      L #s_ISD_ID_Decision.BagIDArray.Decision_Bag_Disposition;
      T #s_Decision_Data.Itm_Data.Process_1.EDS_Decision.Decision_Bag_Disposition;

      L 0;// 0=No decision on current process
      L #s_Decision_Data.Itm_Data.Process_1.EDS_Decision.Decision_Bag_Disposition;
      ==I;
      S #s_Decision_Data.Itm_Data.Process_1.EDS_Decision.No_Decision;
      JC MB10;

      L 1;// 1=Machine alarm
      L #s_Decision_Data.Itm_Data.Process_1.EDS_Decision.Decision_Bag_Disposition;
      ==I;
      S #s_Decision_Data.Itm_Data.Process_1.EDS_Decision.Rejected_Machine;
      JC MB10;

      L 2;// 2=Machine cleared
      L #s_Decision_Data.Itm_Data.Process_1.EDS_Decision.Decision_Bag_Disposition;
      ==I;
      S #s_Decision_Data.Itm_Data.Process_1.EDS_Decision.Cleared_Machine;
      JC MB10;

      L 3;// 3=Machine error / unkown / bag not analyzed
      L #s_Decision_Data.Itm_Data.Process_1.EDS_Decision.Decision_Bag_Disposition;
      ==I;
      S #s_Decision_Data.Itm_Data.Process_1.EDS_Decision.Not_Analyzed;
      JC MB10;

      L 4;// 4=Decision pending
      L #s_Decision_Data.Itm_Data.Process_1.EDS_Decision.Decision_Bag_Disposition;
      ==I;
      S #s_Decision_Data.Itm_Data.Process_1.EDS_Decision.Pending;
      JC MB10;

      L 5;// 5=operator timed out
      L #s_Decision_Data.Itm_Data.Process_1.EDS_Decision.Decision_Bag_Disposition;
      ==I;
      S #s_Decision_Data.Itm_Data.Process_1.EDS_Decision.Timed_Out_Operator;
      JC MB10;

      L 11;//11=operator alarm
      L #s_Decision_Data.Itm_Data.Process_1.EDS_Decision.Decision_Bag_Disposition;
      ==I;
      S #s_Decision_Data.Itm_Data.Process_1.EDS_Decision.Rejected_Operator;
      JC MB10;

      L 12;// 12=operator clear
      L #s_Decision_Data.Itm_Data.Process_1.EDS_Decision.Decision_Bag_Disposition;
      ==I;
      S #s_Decision_Data.Itm_Data.Process_1.EDS_Decision.Cleared_Operator;
      JC MB10;

      L 13;// 13=obvious threat
      L #s_Decision_Data.Itm_Data.Process_1.EDS_Decision.Decision_Bag_Disposition;
      ==I;
      S #s_Decision_Data.Itm_Data.Process_1.EDS_Decision.Obvious_Threat;
      JC MB10;

      L 6;// 6=Machine bag spacing error
      L #s_Decision_Data.Itm_Data.Process_1.EDS_Decision.Decision_Bag_Disposition;
      ==I;
      S #s_Decision_Data.Itm_Data.Process_1.EDS_Decision.Spacing_Error;
      JC MB10;

      L 7;// 7=Forced Reject
      L #s_Decision_Data.Itm_Data.Process_1.EDS_Decision.Decision_Bag_Disposition;
      ==I;
      S #s_Decision_Data.Itm_Data.Process_1.EDS_Decision.Forced_Reject;
      JC MB10;

      SET;// all other result are unknown
      S #s_Decision_Data.Itm_Data.Process_1.EDS_Decision.Not_Analyzed;

MB10:      AN #s_Decision_Data.No_Decision_Expected;
      JCN MB98;

      AN #s_Decision_Data.Valid_LNK_Available;
      JCN MB11;// Item already found, no data reload needed

      A(;
      L #s_Decision_Data.Itm_Data.LNK;
      L 0;
      >I;
      );
      JCN MB12;// If LNK is unknown by EDS, start lookup on pseudo ID

      L #s_Decision_Data.Itm_Data.PEN_ID;
      L "DB_PEN_List".Entries_Present;
      <=I;
      JCN MB98;// If LNK is not in expected range: Abort data attachment

      L "DB_Pending_Record".THIS[#s_Decision_Data.Itm_Data.PEN_ID].PEN_LNK;
      L 0;
      ==I;
      S #s_Decision_Data.No_Decision_Expected;

      AN #s_Decision_Data.No_Decision_Expected;
      JCN MB98;// No HBS record = no screening result expected

      L "DB_Pending_Record".THIS[#s_Decision_Data.Itm_Data.PEN_ID].PEN.LNK;
      L 0;
      >I;
      JCN MB11;

      CALL "FC_Read_ANY_Record"// Read entire LNK record
      (  i_Record_Number             := #s_Decision_Data.Itm_Data.LNK ,
         i_ANY_Data_Record           := "DB_UDT_LNK_Record" ,
         i_ANY_Data                  := #s_Decision_Data.Itm_Data.LNK_Record ,
         i_DB                        := "DB_LNK_List" ,
         i_DB_Event_Num              := #t_DB_Event_Num_Object
      );

MB11:      L #s_Decision_Data.Itm_Data.Pseudo;
      L "DB_Pending_Record".THIS[#s_Decision_Data.Itm_Data.PEN_ID].PEN.PEN_Process_1.Screen_Result.Pseudo_ID;
      ==D;
      JCN MB12;

      L #s_Decision_Data.Itm_Data.PEN_ID;
      L 0;
      >I;
      JCN MB12;

      L "DB_Pending_Record".THIS[#s_Decision_Data.Itm_Data.PEN_ID].PEN.PEN_Process_1.ID_Screening;
      L #i_HBO_ID;
      ==D;
      S #s_Decision_Data.Valid_LNK_Available;
      R #s_Decision_Data.Itm_Data.Process_1.No_Decision_Expected;

      JU MB98;

MB12:      A #s_Decision_Data.Valid_LNK_Available;
      JC MB98;

      A #s_Decision_Data.Itm_Data.Process_1.No_Decision_Expected;
      JC MB99;

      SET;
      S #s_Decision_Data.Inval_LNK_Pseudo_Lookup;

      L DINT#0;
      L #s_Decision_Data.Itm_Data.Pseudo;
      <>D;
      JCN MB98;// If no pseudo available: End bag lookup, else: lookup bag by pseudo

      CALL "FC_PEN_Srch_ID"
      (  i_Pseudo_ID                 := #s_Decision_Data.Itm_Data.Pseudo ,
         o_PEN_ID                    := #s_Decision_Data.Itm_Data.PEN_ID
      );

      L #s_Decision_Data.Itm_Data.PEN_ID;
      L 0;
      >I;
      JCN MB99;

MB50:      AN #s_Decision_Data.Valid_LNK_Available;
      JCN MB98;// If correct LNK not found yet, try next pseudo

MB98:      A #s_Decision_Data.Itm_Data.Process_1.No_Decision_Expected;
      O #s_Decision_Data.No_Decision_Expected;
      AN #s_Decision_Data.Itm_Data.Process_1.EDS_Decision.No_Decision;
      AN #s_Decision_Data.Itm_Data.Process_1.EDS_Decision.Forced_Reject;// We already know the item is no longer present
      AN #s_Decision_Data.Itm_Data.Process_1.EDS_Decision.Not_Analyzed;//With LIC=0 EDS responds Not Analyzed
      JCN MB99;// Unable to find applicable item or item is not pending while decision is present: log event

      CALL "FC_Write_Event"// Screening: Unexpected decision from EDS
      (  i_Message_ID                := 3213 ,
         i_Event_value               := #s_ISD_ID_Decision.BagIDArray.LNK ,
         i_DB_Event_Num              := #t_DB_Event_Num_Object ,
         o_Return_Value              := #t_INT_not_used
      );

MB99:      NOP 0;
NETWORK
TITLE = NA: Upd. PROCESS_1 records (HBS/LIC) upon decision + PackageRep
//Update local bag records to match received decisions
      A #s_OS_New_Decision_Avail;
      A #s_Decision_Data.Valid_LNK_Available;
      JCN NA99;

      AN #s_Decision_Data.Itm_Data.Process_1.No_Decision_Expected;
      JCN NA99;// If no HBS record available: stop receival, else: process

      CALL MOVE
      {value_type := 'Variant'}
      (  IN                          := "DB_Pending_Record".THIS[#s_Decision_Data.Itm_Data.PEN_ID].PEN ,
         OUT                         := #s_Decision_Data.Itm_Data.HBS_Record
      );

      AN #s_Decision_Data.Itm_Data.HBS_Record.PEN_Process_1.Result_Pending;
      O #s_Decision_Data.Itm_Data.HBS_Record.PEN_General.Item_Lost;
      O(;
      L #s_Decision_Data.Itm_Data.HBS_Record.PEN_General.HBA_LNK;
      L #s_Decision_Data.Itm_Data.LNK;
      <>I;
      );
      S #s_Decision_Data.Itm_Data.Process_1.No_Decision_Expected;// No decision expected concluded by HBS record content

      L "DB_Pending_Record".THIS[#s_Decision_Data.Itm_Data.PEN_ID].PEN.LNK;
      L 0;
      ==I;
      S #s_Decision_Data.LIC_Missing;

      A #s_Decision_Data.Itm_Data.Process_1.No_Decision_Expected;
      O #s_Decision_Data.Itm_Data.Process_1.EDS_Decision.No_Decision;
      JC NA23               ;// If process 1 decision expected and present: process, else: make sure PackageReport DB is empty

      A #s_Decision_Data.Itm_Data.Process_1.EDS_Decision.Cleared_Machine;
      AN #s_Decision_Data.Itm_Data.HBS_Record.PEN_Process_1.Machine_Result_Rcvd;
      JCN NA01;
      S #s_Decision_Data.Itm_Data.HBS_Record.PEN_General.Bag_Status.Cleared;
      R #s_Decision_Data.Itm_Data.HBS_Record.PEN_General.Bag_Status.Alarmed;

      L 1;// Update screening status : "CLEAR"
      T #s_Decision_Data.Itm_Data.Process_1.Machine_Result_To_HL;

      SET;
      S #s_Decision_Data.Itm_Data.HBS_Record.PEN_Process_1.Screen_Result.Reached_Screen_Level_1;

      JU NA20;
NA01:      A #s_Decision_Data.Itm_Data.Process_1.EDS_Decision.Rejected_Machine;
      AN #s_Decision_Data.Itm_Data.HBS_Record.PEN_Process_1.Machine_Result_Rcvd;
      JCN NA02;
      S #s_Decision_Data.Itm_Data.HBS_Record.PEN_General.Bag_Status.Alarmed;
      R #s_Decision_Data.Itm_Data.HBS_Record.PEN_General.Bag_Status.Cleared;

      L 2;// Update screening status : "REJECT"
      T #s_Decision_Data.Itm_Data.Process_1.Machine_Result_To_HL;

      SET;
      S #s_Decision_Data.Itm_Data.HBS_Record.PEN_Process_1.Screen_Result.Failed_Screen_Level_1;

      JU NA20;

NA02:      A #s_Decision_Data.Itm_Data.Process_1.EDS_Decision.Not_Analyzed;
      JCN NA04;

      A #s_Decision_Data.Itm_Data.HBS_Record.PEN_General.Bag_Status.NoDecision;
      JCN NA03;
      S #s_Decision_Data.Itm_Data.HBS_Record.PEN_General.Bag_Status.Alarmed;
      R #s_Decision_Data.Itm_Data.HBS_Record.PEN_General.Bag_Status.Cleared;

      L 5;// Suspect
      T #s_Decision_Data.Itm_Data.Process_1.Machine_Result_To_HL;

      SET;
      S #s_Decision_Data.Itm_Data.HBS_Record.PEN_Process_1.Screen_Result.Failed_Screen_Level_1;

      JU NA20;

NA03:      L 5;
      T #s_Decision_Data.Itm_Data.Process_1.Machine_Result_To_HL;

      SET;
      S #s_Decision_Data.Itm_Data.HBS_Record.PEN_General.Bag_Status.Unknown;
//      L     4                    // Not screened/Not Analyzed
//      T     #s_Decision_Data.Itm_Data.HBS_Record.PEN_General.Bag_Status

      JU NA20;

NA04:      A #s_Decision_Data.Itm_Data.Process_1.EDS_Decision.Spacing_Error;
      JCN NA06;

// Check current bag status for result
      A #s_Decision_Data.Itm_Data.HBS_Record.PEN_General.Bag_Status.NoDecision;
      JCN NA05;
      S #s_Decision_Data.Itm_Data.HBS_Record.PEN_General.Bag_Status.Alarmed;
      R #s_Decision_Data.Itm_Data.HBS_Record.PEN_General.Bag_Status.Cleared;

      L 6;
      T #s_Decision_Data.Itm_Data.Process_1.Machine_Result_To_HL;

      SET;
      S #s_Decision_Data.Itm_Data.HBS_Record.PEN_Process_1.Screen_Result.Failed_Screen_Level_1;

      JU NA20;

NA05:      L 5;
      T #s_Decision_Data.Itm_Data.Process_1.Machine_Result_To_HL;

      SET;
      S #s_Decision_Data.Itm_Data.HBS_Record.PEN_General.Bag_Status.Unknown;
//      L     4                    // Not screened/Not Analyzed
//      T     #s_Decision_Data.Itm_Data.HBS_Record.PEN_General.Bag_Status

      JU NA20;

NA06:      A #s_Decision_Data.Itm_Data.Process_1.EDS_Decision.Cleared_Operator;// Evaluate L2 (operator) decision
      AN #s_Decision_Data.Itm_Data.HBS_Record.PEN_Process_1.Operator_Result_Rcvd;
      JCN NA07;// L2 clear
      S #s_Decision_Data.Itm_Data.HBS_Record.PEN_General.Bag_Status.Cleared;
      R #s_Decision_Data.Itm_Data.HBS_Record.PEN_General.Bag_Status.Alarmed;

      L 1;// Update screening status : "CLEAR"
      T #s_Decision_Data.Itm_Data.Process_1.Operator_Result_To_HL;

      SET;
      S #s_Decision_Data.Itm_Data.HBS_Record.PEN_Process_1.Screen_Result.Reached_Screen_Level_2;

      JU NA20;

NA07:      A #s_Decision_Data.Itm_Data.Process_1.EDS_Decision.Rejected_Operator;// L2 fail
      AN #s_Decision_Data.Itm_Data.HBS_Record.PEN_Process_1.Operator_Result_Rcvd;
      JCN NA08;
      S #s_Decision_Data.Itm_Data.HBS_Record.PEN_General.Bag_Status.Alarmed;
      R #s_Decision_Data.Itm_Data.HBS_Record.PEN_General.Bag_Status.Cleared;

      L 6;// Update screening status : "UNCLEARED"
      T #s_Decision_Data.Itm_Data.Process_1.Operator_Result_To_HL;

      SET;
      S #s_Decision_Data.Itm_Data.HBS_Record.PEN_Process_1.Screen_Result.Failed_Screen_Level_2;

      JU NA20;

NA08:      A #s_Decision_Data.Itm_Data.Process_1.EDS_Decision.Timed_Out_Operator;
      AN #s_Decision_Data.Itm_Data.HBS_Record.PEN_Process_1.Operator_Result_Rcvd;
      JCN NA09;
      S #s_Decision_Data.Itm_Data.HBS_Record.PEN_General.Bag_Status.TimeOut;

      L 4;
      T #s_Decision_Data.Itm_Data.Process_1.Operator_Result_To_HL;

      JU NA20;

NA09:      A #s_Decision_Data.Itm_Data.Process_1.EDS_Decision.Pending;
      JCN NA10;// Pending = L1 unclear
      S #s_Decision_Data.Itm_Data.HBS_Record.PEN_General.Bag_Status.Pending;

      L 6;// Update screening status : "UNCLEARED"
      T #s_Decision_Data.Itm_Data.Process_1.Machine_Result_To_HL;

      SET;
      S #s_Decision_Data.Itm_Data.HBS_Record.PEN_Process_1.Screen_Result.Failed_Screen_Level_1;

      JU NA20;

NA10:      A #s_Decision_Data.Itm_Data.Process_1.EDS_Decision.Obvious_Threat;
      AN #s_Decision_Data.Itm_Data.HBS_Record.PEN_Process_1.Operator_Result_Rcvd;
      JCN NA11;// Obvious threat
      S #s_Decision_Data.Itm_Data.HBS_Record.PEN_General.Bag_Status.Alarmed;
      R #s_Decision_Data.Itm_Data.HBS_Record.PEN_General.Bag_Status.Cleared;

      L 6;
      T #s_Decision_Data.Itm_Data.Process_1.Operator_Result_To_HL;

      SET;
      S #s_Decision_Data.Itm_Data.HBS_Record.PEN_Process_1.Screen_Result.Failed_Screen_Level_2;

      JU NA20;

NA11:      A #s_Decision_Data.Itm_Data.Process_1.EDS_Decision.Forced_Reject;
      JCN NA20;// No record updates, only log message

      CALL "FC_Write_Event"// Log: Screening: Force reject on item
      (  i_Message_ID                := 3813 ,
         i_Event_value               := #s_ISD_ID_Decision.BagIDArray.LNK ,
         i_DB_Event_Num              := #t_DB_Event_Num_Object ,
         o_Return_Value              := #t_INT_not_used
      );

      JU NA99;

NA20:      A #s_Decision_Data.Itm_Data.Process_1.EDS_Decision.Cleared_Machine;
      O #s_Decision_Data.Itm_Data.Process_1.EDS_Decision.Rejected_Machine;
      O #s_Decision_Data.Itm_Data.Process_1.EDS_Decision.Not_Analyzed;
      O #s_Decision_Data.Itm_Data.Process_1.EDS_Decision.Spacing_Error;
      O #s_Decision_Data.Itm_Data.Process_1.EDS_Decision.Cleared_Operator;
      O #s_Decision_Data.Itm_Data.Process_1.EDS_Decision.Rejected_Operator;
      O #s_Decision_Data.Itm_Data.Process_1.EDS_Decision.Timed_Out_Operator;
      O #s_Decision_Data.Itm_Data.Process_1.EDS_Decision.Pending;
      O #s_Decision_Data.Itm_Data.Process_1.EDS_Decision.Obvious_Threat;
      JCN NA99;// In case of new data: Update HBS, LIC and send PackageReport

      CALL MOVE
      {value_type := 'Variant'}
      (  IN                          := #s_Decision_Data.Itm_Data.HBS_Record.PEN_Process_1.Screen_Result ,
         OUT                         := "DB_Pending_Record".THIS[#s_Decision_Data.Itm_Data.PEN_ID].PEN.PEN_Process_1.Screen_Result
      );

      CALL MOVE
      {value_type := 'Variant'}
      (  IN                          := #s_Decision_Data.Itm_Data.HBS_Record.PEN_General.Bag_Status ,
         OUT                         := "DB_Pending_Record".THIS[#s_Decision_Data.Itm_Data.PEN_ID].PEN.PEN_General.Bag_Status
      );

      L 0;
      L #s_Decision_Data.Itm_Data.LNK_Record.HBS;
      <I;
      L "DB_HBS_List".Entries_Present;
      <I;
      JCN NA21;

      CALL MOVE
      {value_type := 'Variant'}
      (  IN                          := #s_Decision_Data.Itm_Data.HBS_Record.PEN_General.Bag_Status ,
         OUT                         := "DB_HBS_List".HBS[#s_Decision_Data.Itm_Data.LNK_Record.HBS].PEN_General.Bag_Status
      );

NA21:      A #s_Decision_Data.Itm_Data.HBS_Record.PEN_Process_1.Update_Send;
      JCN NA22               ;// Enable sending of new data if required
      R #s_Decision_Data.Itm_Data.HBS_Record.PEN_Process_1.Update_Send;
      R "DB_Pending_Record".THIS[#s_Decision_Data.Itm_Data.PEN_ID].PEN.PEN_Process_1.Update_Send;

NA22:      CALL "FC_Write_Event"   // Screening pending: Update request from HBO
      (  i_Message_ID                := 3814 ,
         i_Event_value               := #s_Decision_Data.Itm_Data.LNK ,
         i_DB_Event_Num              := #t_DB_Event_Num_Object ,
         o_Return_Value              := #t_INT_not_used
      );

      AN #s_Decision_Data.LIC_Missing;
      JCN NA23;

      CALL "FC_Write_ANY_Record"
      (  i_Record_Number             := #s_Decision_Data.Itm_Data.LNK_Record.LIC ,
         i_ANY_Data_Record           := "DB_UDT_LIC_Record".BIR.Process_1 ,
         i_ANY_Data                  := #s_Decision_Data.Itm_Data.HBS_Record.PEN_Process_1.Screen_Result ,
         i_DB                        := "DB_LIC_List" ,
         i_DB_Event_Num              := #t_DB_Event_Num_Object
      );

      CALL MOVE
      {value_type := 'Variant'}
      (  IN                          := #s_Decision_Data.Itm_Data.HBS_Record.PEN_General.Bag_Status ,
         OUT                         := "DB_LIC_List".LIC[#s_Decision_Data.Itm_Data.LNK_Record.LIC].BIR.Bag_Status
      );

      CALL MOVE
      {value_type := 'Variant'}
      (  IN                          := #s_Decision_Data.Itm_Data.HBS_Record.PEN_Process_1.Screen_Result ,
         OUT                         := "DB_Pending_Record".THIS[#s_Decision_Data.Itm_Data.PEN_ID].PEN.PEN_Process_1.Screen_Result
      );

      CALL MOVE
      {value_type := 'Variant'}
      (  IN                          := #s_Decision_Data.Itm_Data.HBS_Record.PEN_General.Bag_Status ,
         OUT                         := "DB_Pending_Record".THIS[#s_Decision_Data.Itm_Data.PEN_ID].PEN.PEN_General.Bag_Status
      );

NA23:      L #s_Decision_Data.Itm_Data.Process_1.Machine_Result_To_HL;
      L 0;
      >I;
      S #s_Decision_Data.Send_Package_Report;
      R #s_Decision_Data.Package_Report_Sent;
      JCN NA24;
      S "DB_Pending_Record".THIS[#s_Decision_Data.Itm_Data.PEN_ID].PEN.PEN_Process_1.Machine_Result_Rcvd;

      A #s_Decision_Data.Itm_Data.Process_1.EDS_Decision.Not_Analyzed;
      O(;
      A #s_Decision_Data.Itm_Data.Process_1.EDS_Decision.Cleared_Machine;
      AN #s_Decision_Data.Itm_Data.HBS_Record.PEN_Process_1.Screen_Result.Required_Screen_Level_2;
      );
      O #s_Decision_Data.Itm_Data.Process_1.EDS_Decision.Spacing_Error;
      O #s_Decision_Data.Itm_Data.Process_1.EDS_Decision.Forced_Reject;
      JCN NA24;
      R "DB_Pending_Record".THIS[#s_Decision_Data.Itm_Data.PEN_ID].PEN.PEN_Process_1.Result_Pending;

      L #s_Decision_Data.Itm_Data.LNK;
      L 11000;// Bit 11 Process End
      +I;
      T #t_Scn_Event;

      CALL "FC_Write_Event"
      (  i_Message_ID                := 2610 ,
         i_Event_value               := #t_Scn_Event ,
         i_DB_Event_Num              := #t_DB_Event_Num_Object ,
         o_Return_Value              := #t_INT_not_used
      );

NA24:      L #s_Decision_Data.Itm_Data.Process_1.Operator_Result_To_HL;
      L 0;
      >I;
      S #s_Decision_Data.Send_Package_Report;
      R #s_Decision_Data.Package_Report_Sent;
      JCN NA25;
      S "DB_Pending_Record".THIS[#s_Decision_Data.Itm_Data.PEN_ID].PEN.PEN_Process_1.Operator_Result_Rcvd;
      R "DB_Pending_Record".THIS[#s_Decision_Data.Itm_Data.PEN_ID].PEN.PEN_Process_1.Result_Pending;

NA25:      A #s_Decision_Data.Send_Package_Report;
      AN #s_Decision_Data.Package_Report_Sent;
      JCN NA99;

      OPN "DB_Send_FIFO";
      L DBNO;
      T #t_INT_not_used;

      CALL MOVE
      {value_type := 'Variant'}
      (  IN                          := #s_Decision_Data.Itm_Data.HBS_Record.PEN_General.Bag_Status ,
         OUT                         := "DB_Pending_Record".THIS[#s_Decision_Data.Itm_Data.PEN_ID].PEN.PEN_General.Bag_Status
      );

      L "DB_Pending_Record".THIS[#t_PEN_ID].PEN.PEN_General.TRA_LNK;
      L 0;
      <>I;
      JCN NA26;

      CALL "FC_Crt_PendingUpd"
      (  i_ID                        := #i_HBO_ID ,
         i_Data                      := #s_Decision_Data.Itm_Data.PEN_ID ,
         i_TRA_LNK                   := "DB_Pending_Record".THIS[#t_PEN_ID].PEN.PEN_General.TRA_LNK ,
         i_FIFO_PLC_DB_num           := #t_INT_not_used ,
         i_DB_Event_Num              := #t_DB_Event_Num_Object ,
         i_Mess_Type                 := 1
      );

NA26:      AN #s_Decision_Data.LIC_Missing;
      JCN NA97;

      L #s_Decision_Data.Itm_Data.LNK_Record.HBS;
      L 0;
      >I;
      JCN NA97;

      CALL MOVE
      {value_type := 'Variant'}
      (  IN                          := "DB_Pending_Record".THIS[#s_Decision_Data.Itm_Data.PEN_ID].PEN.PEN_General.Bag_Status ,
         OUT                         := "DB_HBS_List".HBS[#s_Decision_Data.Itm_Data.LNK_Record.HBS].PEN_General.Bag_Status
      );

      CALL MOVE
      {value_type := 'Variant'}
      (  IN                          := "DB_Pending_Record".THIS[#s_Decision_Data.Itm_Data.PEN_ID].PEN.PEN_Process_1 ,
         OUT                         := "DB_HBS_List".HBS[#s_Decision_Data.Itm_Data.LNK_Record.HBS].PEN_Process_1
      );

      CALL "FC_Write_ANY_Record"
      (  i_Record_Number             := #s_Decision_Data.Itm_Data.LNK_Record.LIC ,
         i_ANY_Data_Record           := "DB_UDT_LIC_Record".BIR.Process_1 ,
         i_ANY_Data                  := #s_Decision_Data.Itm_Data.HBS_Record.PEN_Process_1.Screen_Result ,
         i_DB                        := "DB_LIC_List" ,
         i_DB_Event_Num              := #t_DB_Event_Num_Object
      );

      CALL "FC_Write_Event"
      (  i_Message_ID                := 1210 , // Send PackageReport: Screening Result
         i_Event_value               := #s_Decision_Data.Itm_Data.LNK ,
         i_DB_Event_Num              := #t_DB_Event_Num_Object ,
         o_Return_Value              := #t_INT_not_used
      );

      JU NA98;

NA97:      CALL "FC_Crt_PackScrnPen"
      (  i_ID                        := #i_HBO_ID ,
         i_PEN_ID                    := #s_Decision_Data.Itm_Data.PEN_ID ,
         i_FIFO_PLC_DB_num           := #t_INT_not_used ,
         i_DB_Event_Num              := #t_DB_Event_Num_Object
      );

NA98:      SET;
      S #s_Decision_Data.Package_Report_Sent;

NA99:      NOP 0;
NETWORK
TITLE = OA: Update PROCESS_1 statisticals upon decision or timeout

      A #s_OS_New_Decision_Avail;
      AN #i_Test_Mode_Active;// Don't update machine decision statisticals in test mode
      JCN OA99;

      A #s_Decision_Data.Itm_Data.Process_1.EDS_Decision.Cleared_Machine;
      JCN OA02;

      L #s_Statisticals.R1.Count_Cleared;
      L 1;
      +I;
      JP OA01;
      L 1;
OA01:      T #s_Statisticals.R1.Count_Cleared;

      JU OA99;

OA02:      A #s_Decision_Data.Itm_Data.Process_1.EDS_Decision.Rejected_Machine;
      JCN OA04;

      L #s_Statisticals.R1.Count_Rejected;
      L 1;
      +I;
      JP OA03;
      L 1;
OA03:      T #s_Statisticals.R1.Count_Rejected;

      JU OA99;

OA04:      A #s_Decision_Data.Itm_Data.Process_1.EDS_Decision.Not_Analyzed;
      JCN OA06;

      L #s_Statisticals.R1.Count_NotAnalyzed;
      L 1;
      +I;
      JP OA05;
      L 1;
OA05:      T #s_Statisticals.R1.Count_NotAnalyzed;

      JU OA99;

OA06:      A #s_Decision_Data.Itm_Data.Process_1.EDS_Decision.Cleared_Operator;// Evaluate L2 (operator) decision
      JCN OA08;// L2 clear

      L #s_Statisticals.R2.Count_Cleared;
      L 1;
      +I;
      JP OA07;
      L 1;
OA07:      T #s_Statisticals.R2.Count_Cleared;

      JU OA99;

OA08:      A #s_Decision_Data.Itm_Data.Process_1.EDS_Decision.Rejected_Operator;// L2 fail
      JCN OA10;

      L #s_Statisticals.R2.Count_Rejected;
      L 1;
      +I;
      JP OA09;
      L 1;
OA09:      T #s_Statisticals.R2.Count_Rejected;

      JU OA99;

OA10:      A #s_Decision_Data.Itm_Data.Process_1.EDS_Decision.Timed_Out_Operator;
      JCN OA12;

      L #s_Statisticals.R2.Count_TimeOut;
      L 1;
      +I;
      JP OA11;
      L 1;
OA11:      T #s_Statisticals.R2.Count_TimeOut;

      JU OA99;

OA12:      A #s_Decision_Data.Itm_Data.Process_1.EDS_Decision.Obvious_Threat;
      JCN OA99;

      L #s_Statisticals.R2.Count_Obvious_Threat;
      L 1;
      +I;
      JP OA13;
      L 1;
OA13:      T #s_Statisticals.R2.Count_Obvious_Threat;

OA99:      NOP 0;
NETWORK
TITLE = PA: Force reject
//When a bag decision is pending while it's no longer required. The bag will be
//force rejected
      CALL #s_FB_HBS_Force_Reject
      (  i_ID                        := #i_HBO_ID ,
         i_Forced_Reject_Ack         := #i_IO_Forced_Reject_Ack ,
         o_Force_Reject              := #o_IO_Force_Reject ,
         o_Pseudo_Code_ForceRej      := #o_IO_Pseud_Code_ForceRej
      );

      A #o_IO_Force_Reject;
      FP #s_FP_Force_Reject;
      JCN PA99;

      L #s_Statisticals.Force_Rejected;
      L 1;
      +I;
      JP PA01;
      L 1;
PA01:      T #s_Statisticals.Force_Rejected;

PA99:      NOP 0;
NETWORK
TITLE = QA: Send and clear statisticals

      A #i_CMD_Send_Stat;
      JCN QA99;

      CALL "FC_Write_Event"
      (  i_Message_ID                := 2001 ,
         i_Event_value               := #s_Statisticals.Bags_Handed_Over ,
         i_DB_Event_Num              := #t_DB_Event_Num_Object ,
         o_Return_Value              := #t_INT_not_used
      );

      CALL "FC_Write_Event"
      (  i_Message_ID                := 2002 ,
         i_Event_value               := #s_Statisticals.Tracking.Positively_Tracked ,
         i_DB_Event_Num              := #t_DB_Event_Num_Object ,
         o_Return_Value              := #t_INT_not_used
      );

      CALL "FC_Write_Event"
      (  i_Message_ID                := 2003 ,
         i_Event_value               := #s_Statisticals.Tracking.Trk_Lost_Result_Pending ,
         i_DB_Event_Num              := #t_DB_Event_Num_Object ,
         o_Return_Value              := #t_INT_not_used
      );

      CALL "FC_Write_Event"
      (  i_Message_ID                := 2004 ,
         i_Event_value               := #s_Statisticals.Tracking.Trk_Lost_No_Result ,
         i_DB_Event_Num              := #t_DB_Event_Num_Object ,
         o_Return_Value              := #t_INT_not_used
      );

      CALL "FC_Write_Event"
      (  i_Message_ID                := 2005 ,
         i_Event_value               := #s_Statisticals.Tracking.Spacing_Error ,
         i_DB_Event_Num              := #t_DB_Event_Num_Object ,
         o_Return_Value              := #t_INT_not_used
      );

      CALL "FC_Write_Event"
      (  i_Message_ID                := 2006 ,
         i_Event_value               := #s_Statisticals.R1.No_Decision_Required ,
         i_DB_Event_Num              := #t_DB_Event_Num_Object ,
         o_Return_Value              := #t_INT_not_used
      );

      CALL "FC_Write_Event"
      (  i_Message_ID                := 2007 ,
         i_Event_value               := #s_Statisticals.R1.Count_Cleared ,
         i_DB_Event_Num              := #t_DB_Event_Num_Object ,
         o_Return_Value              := #t_INT_not_used
      );

      CALL "FC_Write_Event"
      (  i_Message_ID                := 2008 ,
         i_Event_value               := #s_Statisticals.R1.Count_Rejected ,
         i_DB_Event_Num              := #t_DB_Event_Num_Object ,
         o_Return_Value              := #t_INT_not_used
      );

      CALL "FC_Write_Event"
      (  i_Message_ID                := 2009 ,
         i_Event_value               := #s_Statisticals.R2.Count_Cleared ,
         i_DB_Event_Num              := #t_DB_Event_Num_Object ,
         o_Return_Value              := #t_INT_not_used
      );

      CALL "FC_Write_Event"
      (  i_Message_ID                := 2010 ,
         i_Event_value               := #s_Statisticals.R2.Count_Rejected ,
         i_DB_Event_Num              := #t_DB_Event_Num_Object ,
         o_Return_Value              := #t_INT_not_used
      );

      CALL "FC_Write_Event"
      (  i_Message_ID                := 2011 ,
         i_Event_value               := #s_Statisticals.R2.Count_Obvious_Threat ,
         i_DB_Event_Num              := #t_DB_Event_Num_Object ,
         o_Return_Value              := #t_INT_not_used
      );

      CALL "FC_Write_Event"
      (  i_Message_ID                := 2012 ,
         i_Event_value               := #s_Statisticals.R2.Count_TimeOut ,
         i_DB_Event_Num              := #t_DB_Event_Num_Object ,
         o_Return_Value              := #t_INT_not_used
      );

      CALL "FC_Write_Event"
      (  i_Message_ID                := 2013 ,
         i_Event_value               := #s_Statisticals.R1.Count_NotAnalyzed ,
         i_DB_Event_Num              := #t_DB_Event_Num_Object ,
         o_Return_Value              := #t_INT_not_used
      );

      CALL "FC_Write_Event"
      (  i_Message_ID                := 2014 ,
         i_Event_value               := #s_Statisticals.Force_Rejected ,
         i_DB_Event_Num              := #t_DB_Event_Num_Object ,
         o_Return_Value              := #t_INT_not_used
      );

QA99:      NOP 0;
NETWORK
TITLE = RA: Date/Time Master Clock Designator

      CLR;// MV3D is master clock
      = #o_IO_MasterClkDesignator;// No need to send BHS clock

      L #i_IO_Time_Sync_Sec;// Seconds [00..59]
      T #o_IO_Time_Sync_Sec;

      L #i_IO_Time_Sync_Min;// Minutes [00..59]
      T #o_IO_Time_Sync_Min;

      L #i_IO_Time_Sync_Hour;// Time_hours [01..24]
      T #o_IO_Time_Sync_Hour;

      L #i_IO_Time_Sync_Day;// Day of month [1..31]
      T #o_IO_Time_Sync_Day;

      L #i_IO_Time_Sync_Month;// Month [1..31]
      T #o_IO_Time_Sync_Month;

      L #i_IO_Time_Sync_Year;// Year  [0..99]
      T #o_IO_Time_Sync_Year;

NETWORK
TITLE = SA: Object/Section states
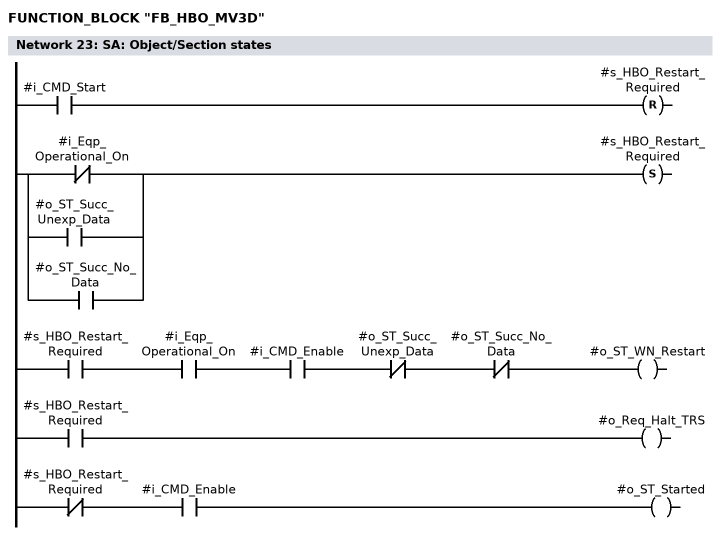

      A #i_CMD_Start;
      R #s_HBO_Restart_Required;

      AN #i_Eqp_Operational_On;
      O #o_ST_Succ_Unexp_Data;
      O #o_ST_Succ_No_Data;
      S #s_HBO_Restart_Required;

      A #s_HBO_Restart_Required;
      A #i_Eqp_Operational_On;
      A #i_CMD_Enable;
      AN #o_ST_Succ_Unexp_Data;
      AN #o_ST_Succ_No_Data;
      = #o_ST_WN_Restart;

      A #s_HBO_Restart_Required;
      = #o_Req_Halt_TRS;

      AN #s_HBO_Restart_Required;
      A #i_CMD_Enable;
      = #o_ST_Started;
NETWORK
TITLE = TA: Copy BHS_ID.BAGIDARRAY (Data) to output
//BHS_ID = BagIDArray + BagIDUpdate
      TAR2 #t_AR2_Store_Restore;// AR2 Store

      L P##i_IO_BHS_ID;// 'area-crossing pointer'
      L #t_Base_Address;// 'relative address'-mask
      +D;
      LAR1;// 'absolute address' Source
      LAR2 P##t_IO_BHS_ID;//  address Destination

      L W[ AR1, P#0.0];// Copy ANY pointer
      T LW[ AR2, P#0.0];// Byte0=$10 (for S7), Byte1=data type
      L W[ AR1, P#2.0];
      T LW[ AR2, P#2.0];// Byte2..3=Repetition factor
      L W[ AR1, P#4.0];
      T LW[ AR2, P#4.0];// Byte4..5=DB number
      L D[ AR1, P#6.0];
      T LD[ AR2, P#6.0];// Byte6=memory area, Byte7..9=Byte,Bit address

      LAR2 #t_AR2_Store_Restore;// AR2 Restore

      CALL BLKMOV
      {blk_type := 'Variant'}
      (  SRCBLK                      := #s_BHS_ID ,
         RET_VAL                     := #t_INT_not_used ,
         DSTBLK                      := #t_IO_BHS_ID
      );

NETWORK
TITLE = UA: Log (1:) BHS.Infeed Bag Process to ApplicationLog
//Log the screening raw data message to the ApplicationLog

      A #o_IO_Inf_Bag_Data_Ready;
      FP #s_FP_IO_Inf_Bag_Data_Ready;
      JCN UA99;

// Clear temp LogMessage using "DB_Outgoing_Msgs".Logging.MessageBody which cleared after usage
      CALL BLKMOV
      {blk_type := 'Variant'}
      (  SRCBLK                      := "DB_Outgoing_Msgs".Logging.MessageBody ,
         RET_VAL                     := #t_INT_not_used ,
         DSTBLK                      := #t_LogMessage
      );

// Add Prefix and separator to log message for indication which message is logged
// '1:' = BHS.Infeed Bag Process
      L '1';
      T #t_LogMessage.Prefix;
      L ':';
      T #t_LogMessage.Separator;

// Convert raw data to a string of ASCII characters
      CALL "FC_Any_Hex_To_Any_ASCII"
      (  i_ANY_Hex_Src               := #s_BHS_ID ,
         i_ANY_ASCII_Dst             := #t_LogMessage.MessageBody ,
         i_DB_Event_Num              := #t_DB_Event_Num_Object
      );

// Load the complete message into Outgoing message buffer
      CALL BLKMOV
      {blk_type := 'Variant'}
      (  SRCBLK                      := #t_LogMessage ,
         RET_VAL                     := #t_INT_not_used ,
         DSTBLK                      := "DB_Outgoing_Msgs".Logging.MessageBody
      );

// Send 2602 ApplicationLog Message
      CALL "FC_Snd_Log_Txt_Msg"
      (  i_ID                        := #i_HBO_ID ,
         i_Event_value               := 1
      );

UA99:      NOP 0;

NETWORK
TITLE = UB: Log (2:) EDS.Exit Bag Process to ApplicationLog
//Log the screening raw data message to the ApplicationLog

      A #i_IO_Receive_Data_Outf;
      FP #s_FP_IO_Receive_Data_Outf;
      JCN UB99;

// Clear temp LogMessage using "DB_Outgoing_Msgs".Logging.MessageBody which cleared after usage
      CALL BLKMOV
      {blk_type := 'Variant'}
      (  SRCBLK                      := "DB_Outgoing_Msgs".Logging.MessageBody ,
         RET_VAL                     := #t_INT_not_used ,
         DSTBLK                      := #t_LogMessage
      );

// Add Prefix and separator to log message for indication which message is logged
// '2:' = EDS.Exit Bag Process
      L '2';
      T #t_LogMessage.Prefix;
      L ':';
      T #t_LogMessage.Separator;

// Convert raw data to a string of ASCII characters
      CALL "FC_Any_Hex_To_Any_ASCII"
      (  i_ANY_Hex_Src               := #s_ISD_ID_Tracking ,
         i_ANY_ASCII_Dst             := #t_LogMessage.MessageBody ,
         i_DB_Event_Num              := #t_DB_Event_Num_Object
      );

// Load the complete message into Outgoing message buffer
      CALL BLKMOV
      {blk_type := 'Variant'}
      (  SRCBLK                      := #t_LogMessage ,
         RET_VAL                     := #t_INT_not_used ,
         DSTBLK                      := "DB_Outgoing_Msgs".Logging.MessageBody
      );

// Send 2602 ApplicationLog Message
      CALL "FC_Snd_Log_Txt_Msg"
      (  i_ID                        := #i_HBO_ID ,
         i_Event_value               := 2
      );

UB99:      NOP 0;

NETWORK
TITLE = UC: Log (3:) EDS.Screening Result to ApplicationLog
//Log the screening raw data message to the ApplicationLog

      A #i_IO_Decision_Available;
      FP #s_FP_IO_Decision_Available;
      JCN UC99;

// Clear temp LogMessage using "DB_Outgoing_Msgs".Logging.MessageBody which cleared after usage
      CALL BLKMOV
      {blk_type := 'Variant'}
      (  SRCBLK                      := "DB_Outgoing_Msgs".Logging.MessageBody ,
         RET_VAL                     := #t_INT_not_used ,
         DSTBLK                      := #t_LogMessage
      );

// Add Prefix and separator to log message for indication which message is logged
// '3:' = EDS.Screening Result
      L '3';
      T #t_LogMessage.Prefix;
      L ':';
      T #t_LogMessage.Separator;

// Convert raw data to a string of ASCII characters
      CALL "FC_Any_Hex_To_Any_ASCII"
      (  i_ANY_Hex_Src               := #s_ISD_ID_Decision ,
         i_ANY_ASCII_Dst             := #t_LogMessage.MessageBody ,
         i_DB_Event_Num              := #t_DB_Event_Num_Object
      );

// Load the complete message into Outgoing message buffer
      CALL BLKMOV
      {blk_type := 'Variant'}
      (  SRCBLK                      := #t_LogMessage ,
         RET_VAL                     := #t_INT_not_used ,
         DSTBLK                      := "DB_Outgoing_Msgs".Logging.MessageBody
      );

// Send 2602 ApplicationLog Message
      CALL "FC_Snd_Log_Txt_Msg"
      (  i_ID                        := #i_HBO_ID ,
         i_Event_value               := 3
      );

UC99:      NOP 0;

NETWORK
TITLE = UD: Log (4:) BHS.ForcedReject to ApplicationLog
//Log the screening raw data message to the ApplicationLog

      A #o_IO_Force_Reject;
      FP #s_FP_IO_Force_Reject;
      JCN UD99;

// Clear temp LogMessage using "DB_Outgoing_Msgs".Logging.MessageBody which cleared after usage
      CALL BLKMOV
      {blk_type := 'Variant'}
      (  SRCBLK                      := "DB_Outgoing_Msgs".Logging.MessageBody ,
         RET_VAL                     := #t_INT_not_used ,
         DSTBLK                      := #t_LogMessage
      );

// Add Prefix and separator to log message for indication which message is logged
// '4:' = BHS.ForcedReject
      L '4';
      T #t_LogMessage.Prefix;
      L ':';
      T #t_LogMessage.Separator;

// Convert raw data to a string of ASCII characters
      CALL "FC_Any_Hex_To_Any_ASCII"
      (  i_ANY_Hex_Src               := #o_IO_Pseud_Code_ForceRej ,
         i_ANY_ASCII_Dst             := #t_LogMessage.MessageBody ,
         i_DB_Event_Num              := #t_DB_Event_Num_Object
      );

// Load the complete message into Outgoing message buffer
      CALL BLKMOV
      {blk_type := 'Variant'}
      (  SRCBLK                      := #t_LogMessage ,
         RET_VAL                     := #t_INT_not_used ,
         DSTBLK                      := "DB_Outgoing_Msgs".Logging.MessageBody
      );

// Send 2602 ApplicationLog Message
      CALL "FC_Snd_Log_Txt_Msg"
      (  i_ID                        := #i_HBO_ID ,
         i_Event_value               := 4
      );

UD99:      NOP 0;

NETWORK
TITLE = UE: Log (5:) EDS.ForcedReject to ApplicationLog
//Log the screening raw data message to the ApplicationLog

      A #i_IO_Forced_Reject_Ack;
      FP #s_FP_IO_Forced_Reject_Ack;
      JCN UE99;

// Clear temp LogMessage using "DB_Outgoing_Msgs".Logging.MessageBody which cleared after usage
      CALL BLKMOV
      {blk_type := 'Variant'}
      (  SRCBLK                      := "DB_Outgoing_Msgs".Logging.MessageBody ,
         RET_VAL                     := #t_INT_not_used ,
         DSTBLK                      := #t_LogMessage
      );

// Add Prefix and separator to log message for indication which message is logged
// '5:' = EDS.ForcedReject
      L '5';
      T #t_LogMessage.Prefix;
      L ':';
      T #t_LogMessage.Separator;

// Convert raw data to a string of ASCII characters
      CALL "FC_Any_Hex_To_Any_ASCII"
      (  i_ANY_Hex_Src               := #s_ISD_ID_Decision ,
         i_ANY_ASCII_Dst             := #t_LogMessage.MessageBody ,
         i_DB_Event_Num              := #t_DB_Event_Num_Object
      );

// Load the complete message into Outgoing message buffer
      CALL BLKMOV
      {blk_type := 'Variant'}
      (  SRCBLK                      := #t_LogMessage ,
         RET_VAL                     := #t_INT_not_used ,
         DSTBLK                      := "DB_Outgoing_Msgs".Logging.MessageBody
      );

// Send 2602 ApplicationLog Message
      CALL "FC_Snd_Log_Txt_Msg"
      (  i_ID                        := #i_HBO_ID ,
         i_Event_value               := 5
      );

UE99:      NOP 0;
END_FUNCTION_BLOCK


